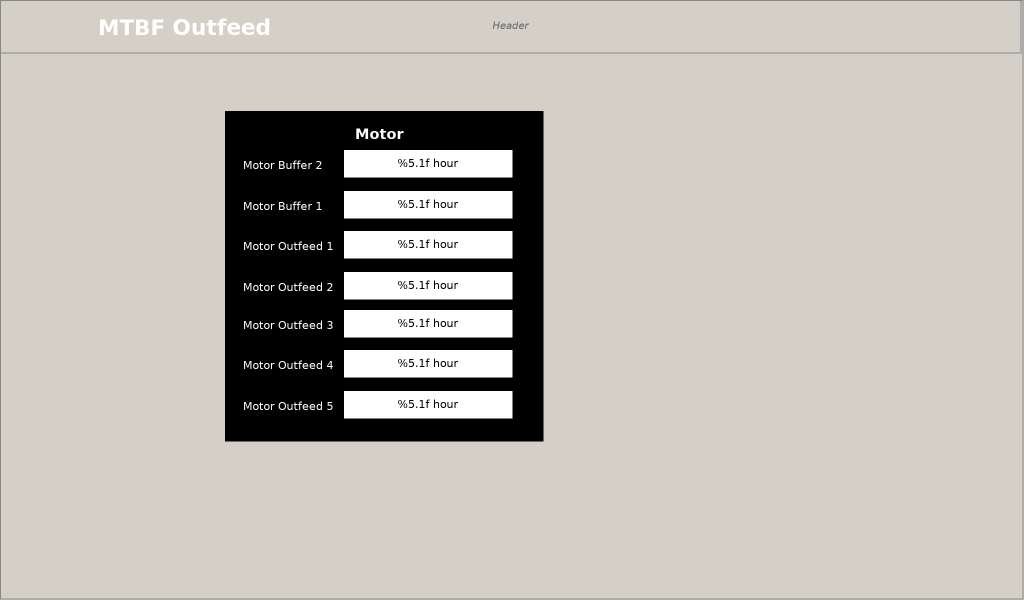
VISUALIZATION MTBF_Outfeed  // 1024x600
    Frame (0,-2 1021x55)
        shows Header()
    Label (95,15 250x25), "MTBF Outfeed"
    RoundedRectangle (225,111 318x330)
    Label (243,114 273x40), "Motor"
    Label (240,148 103x35), "Motor Buffer 2"
    RoundedRectangle (343,149 170x29), "%5.1f hour", text variable: InputOutput_GVL.MTBF_Motor[1]
    Label (240,189 103x35), "Motor Buffer 1"
    RoundedRectangle (343,190 170x29), "%5.1f hour", text variable: InputOutput_GVL.MTBF_Motor[2]
    Label (240,229 103x35), "Motor Outfeed 1"
    RoundedRectangle (343,230 170x29), "%5.1f hour", text variable: InputOutput_GVL.MTBF_Motor[3]
    Label (240,270 103x35), "Motor Outfeed 2"
    RoundedRectangle (343,271 170x29), "%5.1f hour", text variable: InputOutput_GVL.MTBF_Motor[4]
    Label (240,308 103x35), "Motor Outfeed 3"
    RoundedRectangle (343,309 170x29), "%5.1f hour", text variable: InputOutput_GVL.MTBF_Motor[5]
    Label (240,348 103x35), "Motor Outfeed 4"
    RoundedRectangle (343,349 170x29), "%5.1f hour", text variable: InputOutput_GVL.MTBF_Motor[6]
    Label (240,389 103x35), "Motor Outfeed 5"
    RoundedRectangle (343,390 170x29), "%5.1f hour", text variable: InputOutput_GVL.MTBF_Motor[7]
END_VISUALIZATION

(* stored: Version 1.1.0.1, ProductVersion 3.1.4024.12
   Visu MTBF_Outfeed: Id {a2e325c5-5fb0-4613-8082-21e35bd962d3} *)
